	FUNCTION_BLOCK FB 193
	TITLE =G093M BELT CONVEYOR 4300 GERM
	//COPYRIGHT:    (C) 2009  BUHLER AG, CH-9240 UZWIL, SWITZERLAND
	//
	//PRODUCT:      WinCoS_BIW01_09
	//
	//TITLE:        BELT CONVEYOR 4300 GERM
	//                Machine group control
	//                Maschinengruppensteuerung
	//
	//--------------------------------------------------------------------------------
	//
	//IDENT:        AUTHOR:             DEPT:                              DATE:
	//
	//P01_FB193.1.0 K.Renz              CSB41                              13.Jan.2010
	//             1st Release
	//
	//--------------------------------------------------------------------------------
	//
	//PURPOSE:
	//
	//MANUAL :
	//
	//RESTRICTIONS:
	//
	//--------------------------------------------------------------------------------
	AUTHOR  : KR
	FAMILY  : USW
	VERSION : 9.9


	VAR
	  Gr       : FB10;	//Standard interface to group
	  InOutValue1    : DINT; //Data for user
	  InOutValue2    : DINT; //Data for user
	  OutWayConflict : BOOL;	//Data for user
	  OutSelectionOk : BOOL;	//Data for user
	  CmdNewValue : BOOL;	//Data for user
	  CmdNewJob   : BOOL;	//Data for user
	  OutCodeOK   : BOOL;	//Data for user
	  InEndOfJob  : BOOL ;	//Data for user
	  staWayOk      : BOOL ;	//Data for user
	  EdgeStartRelease : BOOL ;	//Data for user
	  USW8  : BOOL;	//Data for user
	  USW9 : BOOL;	//Data for user
	  USW10: BOOL;	//Data for user
	  USW11: BOOL;	//Data for user
	  USW12: BOOL;	//Data for user
	  USW13: BOOL;	//Data for user
	  USW14: BOOL;	//Data for user
	  USW15: BOOL;	//Data for user
	     #A_1921_MXZ01MA : FB1002;   // Motor+6DI
	     #A_1921_QXV31 : FB13;   // VLS
	     #A_1921_BFT07 : FB84;   // SubType FB14: DigInpCont
	END_VAR
	VAR_TEMP
	   tmpEnable		: BOOL;
	   tmpFlag  		: BOOL;
	   tmpCmdNext		: BOOL;
	   tmpLocal  		: BOOL;
	   tmpAspOk  		: BOOL;
	   tmpHWStop 		: BOOL;
	   tmpInstanzDBNo       : INT ;
	END_VAR
	BEGIN
	NETWORK
	TITLE =
	NETWORK
	TITLE =Read command from group control
	//Parameter
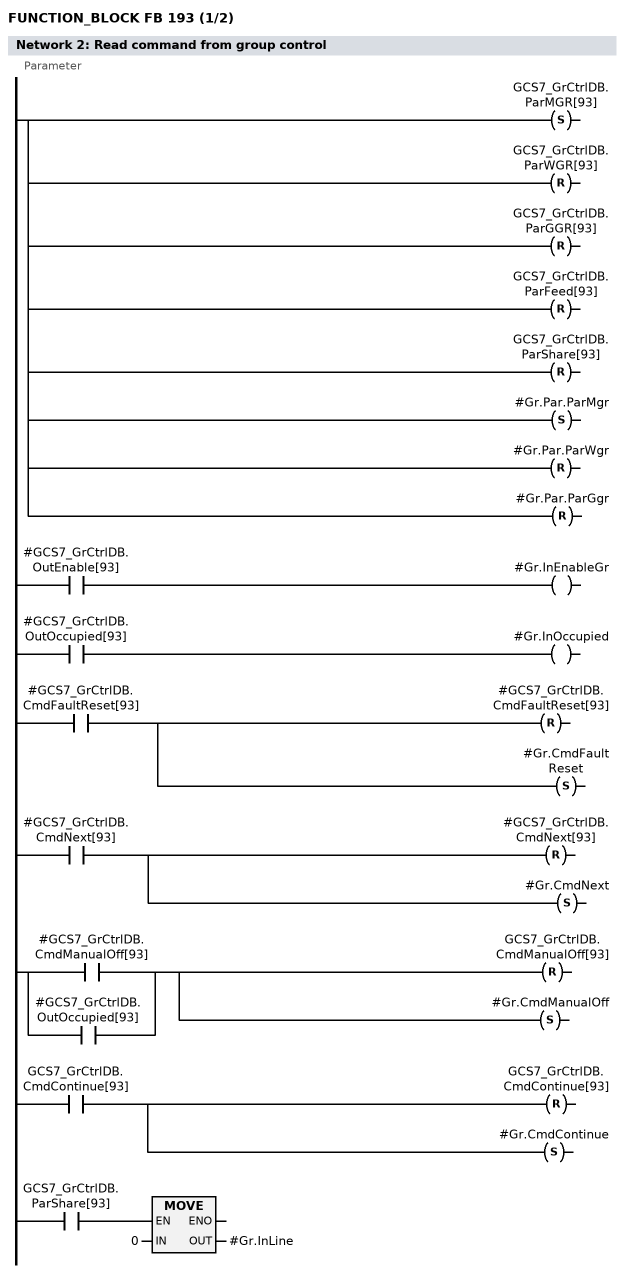
	      SET;
	      S   GCS7_GrCtrlDB.ParMGR[93];
	      R   GCS7_GrCtrlDB.ParWGR[93];
	      R   GCS7_GrCtrlDB.ParGGR[93];
	      R   GCS7_GrCtrlDB.ParFeed[93];
	      R   GCS7_GrCtrlDB.ParShare[93];
	      S   #Gr.Par.ParMgr;
	      R   #Gr.Par.ParWgr;
	      R   #Gr.Par.ParGgr;
	//Command
	      U   #GCS7_GrCtrlDB.OutEnable[93];
	      =   #Gr.InEnableGr;
	      U   #GCS7_GrCtrlDB.OutOccupied[93];
	      =   #Gr.InOccupied;
	      U   #GCS7_GrCtrlDB.CmdFaultReset[93];
	      R   #GCS7_GrCtrlDB.CmdFaultReset[93];
	      S   #Gr.CmdFaultReset;
	      U  #GCS7_GrCtrlDB.CmdNext[93];
	      R   #GCS7_GrCtrlDB.CmdNext[93];
	      S   #Gr.CmdNext;
	      U   #GCS7_GrCtrlDB.CmdManualOff[93];
	      O   #GCS7_GrCtrlDB.OutOccupied[93];
	      R   GCS7_GrCtrlDB.CmdManualOff[93];
	      S   #Gr.CmdManualOff;
	      U  GCS7_GrCtrlDB.CmdContinue[93];
	      R   GCS7_GrCtrlDB.CmdContinue[93];
	      S   #Gr.CmdContinue;
	//Init Line Number
	      U   GCS7_GrCtrlDB.ParShare[93];
	      SPBN WE00;
	      L     0;
	      T     #Gr.InLine;
	WE00: NOP   0;
	NETWORK
	TITLE =Call Methode Control
	// 1. Handle Interface PCControl
	// 2. Prepare mode --> ModePassive,ModeActive,ModeIdling
	// 3. Reset global flags of the group
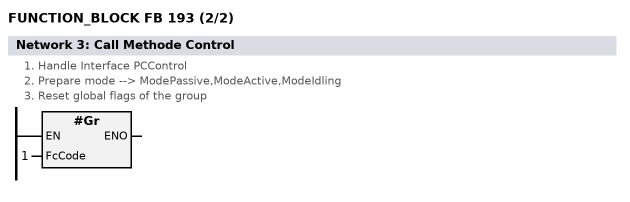
	      CALL #Gr (
	           FcCode                   := 1);
	NETWORK
	TITLE =Restart Idling Time
		L  #Gr.Par.ParIdling;
		L  2;
		>=I;
		SPB IdTm;
		T  #Gr.Par.ParIdling;
	IdTm:   NOP 0;
	      CLR;
	      S    #Gr.CmdRestartIdling;
	NETWORK
	TITLE =Prepare global flags
	NETWORK
	TITLE =Set Pattern (Target position)
	NETWORK
	TITLE =Interlocking WayOk
	//
	NETWORK
	TITLE =Interlocking Autostart
		CLR;
		R   #Gr.OutAutostart;
	NETWORK
	TITLE =Interlocking Enable
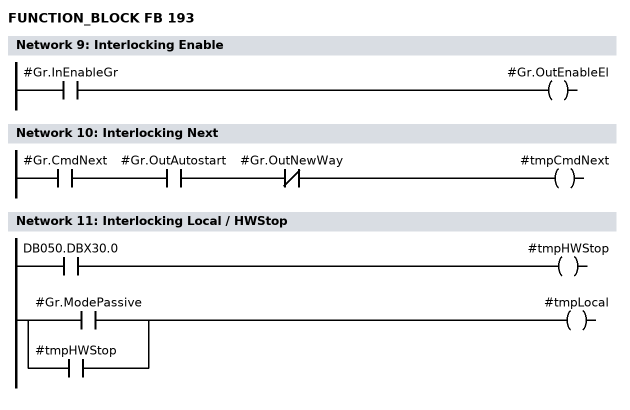
	      U     #Gr.InEnableGr;
	      =     #Gr.OutEnableEl;

	NETWORK
	TITLE =Interlocking Next
	      U     #Gr.CmdNext;
	      U     #Gr.OutAutostart;
	      UN    #Gr.OutNewWay;
	      =    #tmpCmdNext;

	NETWORK
	TITLE =Interlocking Local / HWStop
	      U    DB050.DBX30.0;
	      =    #tmpHWStop;

	      U    #Gr.ModePassive;
	      O    #tmpHWStop;
	      =    #tmpLocal;

	NETWORK
	TITLE =Interlocking Start Warning
	      NOP 0;
	//- Restart after fault --
	      U     #Gr.CmdFaultReset;
	      U     #Gr.VarFault;
	      S       "SYS_StartWarningDB".Area[1].CmdResetStartWarning;
	//- Run Timer --
	      AUF "G093M";
	      CALL  FB100 , DB100(
	       InModeHigher :=FALSE,
	       InArea     :=1,
	       InEnable   :=#Gr.OutEnableEl,
	       InLocal    :=#tmpLocal,
	       InStarted  :=#Gr.VarStarted,
	       InCmdNext  :=#tmpCmdNext,
	       OutCmdNext :=#tmpCmdNext,
	       OutStartwarning:=#Gr.VarStartWarning);
	//- Store Startwarning done  --
	//- Reset Autostart --
	      U     "SYS_StartWarningDB".TmpArea.OutStartReleaseRunningL;
	      FN    #EdgeStartRelease;
	      U     #Gr.VarFault;
	      R     #Gr.OutAutostart;
	NETWORK
	TITLE ==A-1921-BFT07 : STOWING DETECTOR DISCHARGE
	NOP 0;
	//-InLocal---
	      U     #tmpLocal;
	      =     #A_1921_BFT07.InLocal;
	//
	//-Monitoring---
	      CLR;
	      =      #A_1921_BFT07.InMonCovered;
	      SET;
	      =      #A_1921_BFT07.InMonUncovered;
	//
	//-PreAlarm---
	      CLR;
	      =      #A_1921_BFT07.InPreAlarmCovered;
	      CLR;
	      =      #A_1921_BFT07.InPreAlarmUncovered;
	//
	//-Additional commands---
	//      CLR
	//      S     #A_1921_BFT07.CmdRunTimeOutTime
	//
	//-Read inputs---
	      UN    E 1109.0;
	      =     #A_1921_BFT07.InpCovered;
	      U   DB050.DBX31.0;
	      =     #A_1921_BFT07.InHWStop;
	       U     PLC_DPInfo.Master[1].SlavesError[111];
	       =       #A_1921_BFT07.InDPFault;
	//
	//-Set Parameters---
	//
	//-Call object control---
	      CALL  #A_1921_BFT07;
	//
	//-Write outputs---
	NETWORK
	TITLE ==A-1921-MXZ01MA : BELT CONVEYOR 4300
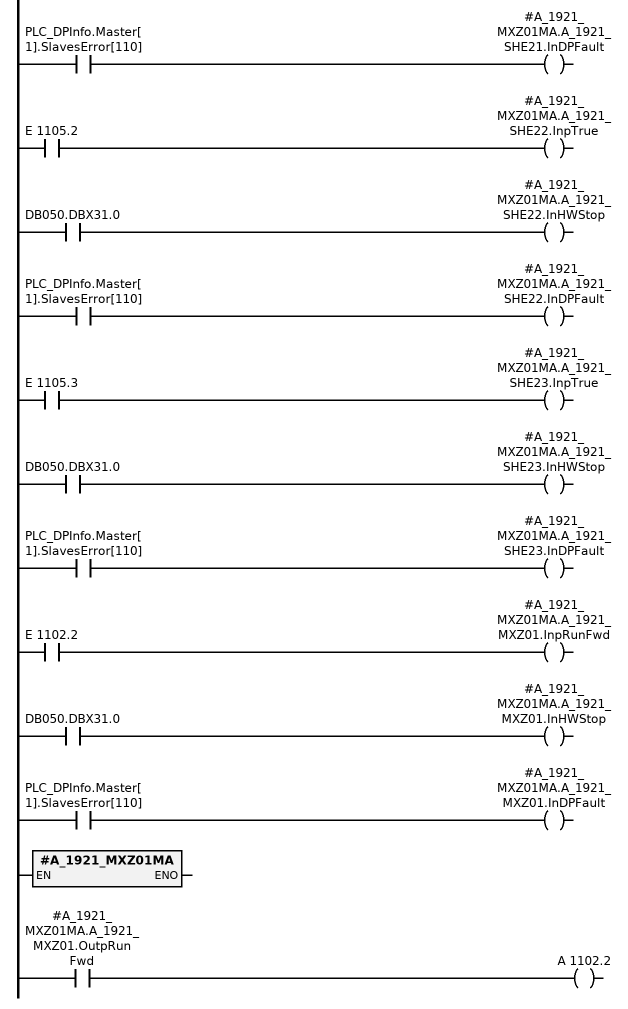
	NOP 0;
	//-InLocal---
	      U     #tmpLocal;
	      =     #A_1921_MXZ01MA.Ma.InLocal;
	//
	//-Interlocking---
	      UN    #A_1921_BFT07.StFault;
	      U     #Gr.OutEnableEl;
	      =     #A_1921_MXZ01MA.Ma.InEnableFwd;
	//
	      U    #tmpCmdNext;
	      S     #A_1921_MXZ01MA.Ma.CmdNext;
	//
	      U     #Gr.OutSeqStop;
	      =     #A_1921_MXZ01MA.Ma.InSeqStop;
	//
	//=Values and commands of elements===
	//-=A-1921-SHE20---
	//      CLR
	//      S     #A_1921_MXZ01MA.A_1921_SHE20.CmdRunTimeOutTime
	//-=A-1921-BSA13---
	//      CLR
	//      S     #A_1921_MXZ01MA.A_1921_BSA13.CmdRunTimeOutTime
	//-=A-1921-BZS14/15---
	//      CLR
	//      S     #A_1921_MXZ01MA.A_1921_BZS14_15.CmdRunTimeOutTime
	//-=A-1921-SHE21---
	//      CLR
	//      S     #A_1921_MXZ01MA.A_1921_SHE21.CmdRunTimeOutTime
	//-=A-1921-SHE22---
	//      CLR
	//      S     #A_1921_MXZ01MA.A_1921_SHE22.CmdRunTimeOutTime
	//-=A-1921-SHE23---
	//      CLR
	//      S     #A_1921_MXZ01MA.A_1921_SHE23.CmdRunTimeOutTime
	//
	//-Read inputs of elements---
	      U     E 1105.0;
	      =     #A_1921_MXZ01MA.A_1921_SHE20.InpTrue;
	      U   DB050.DBX31.0;
	      =     #A_1921_MXZ01MA.A_1921_SHE20.InHWStop;
	       U     PLC_DPInfo.Master[1].SlavesError[110];
	       =       #A_1921_MXZ01MA.A_1921_SHE20.InDPFault;
	      U     E 1109.1;
	      =     #A_1921_MXZ01MA.A_1921_BSA13.InpTrue;
	      U   DB050.DBX31.0;
	      =     #A_1921_MXZ01MA.A_1921_BSA13.InHWStop;
	       U     PLC_DPInfo.Master[1].SlavesError[111];
	       =       #A_1921_MXZ01MA.A_1921_BSA13.InDPFault;
	      U     E 1109.2;
	      =     #A_1921_MXZ01MA.A_1921_BZS14_15.InpTrue;
	      U   DB050.DBX31.0;
	      =     #A_1921_MXZ01MA.A_1921_BZS14_15.InHWStop;
	       U     PLC_DPInfo.Master[1].SlavesError[111];
	       =       #A_1921_MXZ01MA.A_1921_BZS14_15.InDPFault;
	      U     E 1105.1;
	      =     #A_1921_MXZ01MA.A_1921_SHE21.InpTrue;
	      U   DB050.DBX31.0;
	      =     #A_1921_MXZ01MA.A_1921_SHE21.InHWStop;
	       U     PLC_DPInfo.Master[1].SlavesError[110];
	       =       #A_1921_MXZ01MA.A_1921_SHE21.InDPFault;
	      U     E 1105.2;
	      =     #A_1921_MXZ01MA.A_1921_SHE22.InpTrue;
	      U   DB050.DBX31.0;
	      =     #A_1921_MXZ01MA.A_1921_SHE22.InHWStop;
	       U     PLC_DPInfo.Master[1].SlavesError[110];
	       =       #A_1921_MXZ01MA.A_1921_SHE22.InDPFault;
	      U     E 1105.3;
	      =     #A_1921_MXZ01MA.A_1921_SHE23.InpTrue;
	      U   DB050.DBX31.0;
	      =     #A_1921_MXZ01MA.A_1921_SHE23.InHWStop;
	       U     PLC_DPInfo.Master[1].SlavesError[110];
	       =       #A_1921_MXZ01MA.A_1921_SHE23.InDPFault;
	      U     E 1102.2;
	      =     #A_1921_MXZ01MA.A_1921_MXZ01.InpRunFwd;
	      U   DB050.DBX31.0;
	      =     #A_1921_MXZ01MA.A_1921_MXZ01.InHWStop;
	       U     PLC_DPInfo.Master[1].SlavesError[110];
	       =       #A_1921_MXZ01MA.A_1921_MXZ01.InDPFault;
	//
	//-Set Parameters---
	//
	//-Call object control---
	      CALL  #A_1921_MXZ01MA;
	//
	//-Write outputs---
	      U     #A_1921_MXZ01MA.A_1921_MXZ01.OutpRunFwd;
	      =     A 1102.2;
	NETWORK
	TITLE ==A-1921-QXV31 : BALL VALVE SPRAY WATER OPEN
	NOP 0;
	//-InLocal---
	      U     #tmpLocal;
	      =     #A_1921_QXV31.InLocal;
	//
	//-Interlocking---
	      U A_1921_MXZ01MA.Ma.StStartedFwd;
	         =     #A_1921_QXV31.InEnableHN;
	         NOT;
	         =     #A_1921_QXV31.InEnableLN;
	//
	         SET;
	         S     #A_1921_QXV31.CmdNext;
	//
	      U     #Gr.OutSeqStop;
	      =     #A_1921_QXV31.InSeqStop;
	//
	//-Read inputs---
	      UN   #A_1921_QXV31.OutpHN;
	      =     #A_1921_QXV31.InpLN;
	      U   #A_1921_QXV31.OutpHN;
	      =     #A_1921_QXV31.InpHN;
	      U   DB050.DBX31.2;
	      =     #A_1921_QXV31.InHWStop;
	       U     PLC_DPInfo.Master[1].SlavesError[111];
	       =       #A_1921_QXV31.InDPFault;
	//
	//-Set Parameters---
	//
	//-Call object control---
	      CALL  #A_1921_QXV31;
	//
	//-Write outputs---
	      U     #A_1921_QXV31.OutpHN;
	      =     A 1108.2;
	NETWORK
	TITLE =Test Fault
	      U     #A_1921_BFT07.StFault;
	      O     #A_1921_MXZ01MA.Ma.StFault;
	      O     #A_1921_QXV31.StFault;
	      =     #Gr.VarFault;
	NETWORK
	TITLE =Test Warning
	      CLR;
	      =     #Gr.OutWarning;
	NETWORK
	TITLE =Test Stopped
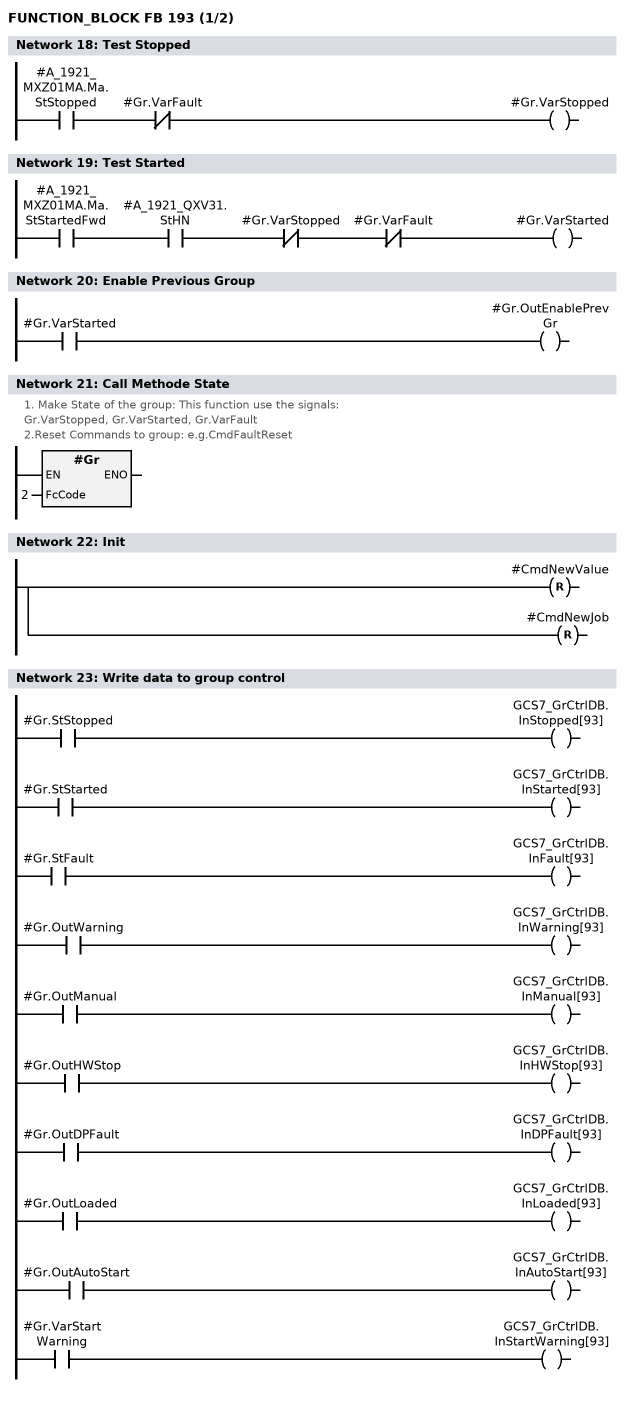
	      U     #A_1921_MXZ01MA.Ma.StStopped;
	      UN   #Gr.VarFault;
	      =     #Gr.VarStopped;
	NETWORK
	TITLE =Test Started
	      U     #A_1921_MXZ01MA.Ma.StStartedFwd;
	      U     #A_1921_QXV31.StHN;
	      UN  #Gr.VarStopped;
	      UN  #Gr.VarFault;
	      =     #Gr.VarStarted;
	NETWORK
	TITLE =Enable Previous Group
	      U    #Gr.VarStarted;
	      =     #Gr.OutEnablePrevGr;
	NETWORK
	TITLE =Call Methode State
	//1. Make State of the group: This function use the signals:
	//        Gr.VarStopped, Gr.VarStarted, Gr.VarFault
	//2.Reset Commands to group: e.g.CmdFaultReset
	      CALL #Gr (
	           FcCode                   := 2);
	NETWORK
	TITLE =Init
	      SET;
	      R    #CmdNewValue;
	      R    #CmdNewJob;
	NETWORK
	TITLE =Write data to group control
	      U   #Gr.StStopped;
	      =   GCS7_GrCtrlDB.InStopped[93];
	      U   #Gr.StStarted;
	      =   GCS7_GrCtrlDB.InStarted[93];
	      U   #Gr.StFault;
	      =   GCS7_GrCtrlDB.InFault[93];
	      U   #Gr.OutWarning;
	      =   GCS7_GrCtrlDB.InWarning[93];
	      U   #Gr.OutManual;
	      =   GCS7_GrCtrlDB.InManual[93];
	      U   #Gr.OutHWStop;
	      =   GCS7_GrCtrlDB.InHWStop[93];
	      U   #Gr.OutDPFault;
	      =   GCS7_GrCtrlDB.InDPFault[93];
	      U   #Gr.OutLoaded;
	      =   GCS7_GrCtrlDB.InLoaded[93];
	      U   #Gr.OutAutoStart;
	      =   GCS7_GrCtrlDB.InAutoStart[93];
	      U   #Gr.VarStartWarning;
	      =   GCS7_GrCtrlDB.InStartWarning[93];
	NETWORK
	TITLE =End of block
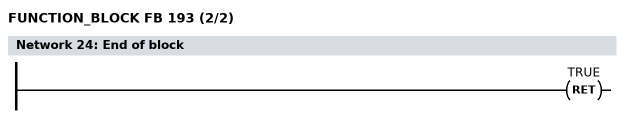

	BE

	END_FUNCTION_BLOCK
